# EPICS substitutions: examples/test/el6080/ecmcEL6080_app_floats.substitutions
file "ecmcEL6080_app_floats.template"
{
  pattern {EC_TYPE}
          {F32    }
          {F64    }
}
